Fanuc TP program (LS listing): TWICE.LS

/PROG  TWICE
/ATTR
OWNER		= MNEDITOR;
COMMENT		= "Twice";
PROG_SIZE	= 0;
CREATE		= DATE 26-01-01  TIME 00:00:00;
MODIFIED	= DATE 26-01-01  TIME 00:00:00;
FILE_NAME	= ;
VERSION		= 0;
LINE_COUNT	= 6;
MEMORY_SIZE	= 0;
PROTECT		= READ_WRITE;
TCD:  STACK_SIZE	= 0,
      TASK_PRIORITY	= 50,
      TIME_SLICE	= 0,
      BUSY_LAMP_OFF	= 0,
      ABORT_REQUEST	= 0,
      PAUSE_REQUEST	= 0;
DEFAULT_GROUP	= 1,*,*,*,*;
CONTROL_CODE	= 00000000 00000000;
/MN
   1:  !RAPID PointProbe.Twice ;
   2:  PR[99]=PR[98]    ;
   3:  CALL PICKAT    ;
   4:  PR[99]=PR[98]    ;
   5:  PR[99,1]=PR[99,1]+30    ;
   6:  CALL PICKAT    ;
/POS
/END
